ABB RAPID module: Part_8.mod

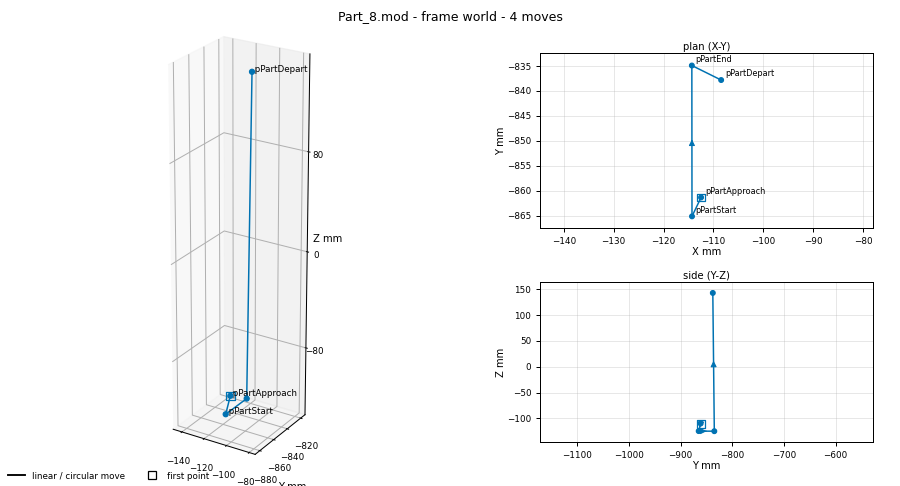
[picture p0: tool path of Part_8.mod in frame world, 4 of 9 moves have a stored position in this frame; points joined in program order, loops and branches not executed]
MODULE Part_8
  ! ------------------------------------------------------------------
  ! Single-part welding template
  !
  ! Purpose:
  !   - Run one part only (no multi-part branching)
  !   - Keep nozzle cleaning and BullsEye tool check available
  !   - Provide a copy/paste starting point for new part files
  !
  ! Dependencies:
  !   - LogicZ (home/safe/pounce positions + rTC2013)
  !   - BE_User1 (BECheckToolb for BullsEye)
  !   - mTSC (optional torch cleaner if you prefer MechCleanGun)
  ! ------------------------------------------------------------------

  PERS bool bUseTorchClean := TRUE;
  PERS bool bUseBullseye := TRUE;

  ! Placeholder weld/seam data for the template. Replace with real values.
  TASK PERS welddata weldPart := [0,0,[1,0,0,0,0,0,0,0,0],[0,0,0,0,0,0,0,0,0]];
  TASK PERS seamdata seamPart := [1,1,[1,0,0,0,0,0,0,0,0],0,0,0,0,0,[0,0,0,0,0,0,0,0,0],0,0,[0,0,0,0,0,0,0,0,0],0,0,[0,0,0,0,0,0,0,0,0],0];

  ! Placeholder targets for the weld path. Replace with taught points.
  CONST robtarget pPartApproach := [[-112.47,-861.36,-110.12],[0.220582,0.688805,-0.67554,-0.143307],[-1,-1,-2,0],[9E+09,9E+09,9E+09,9E+09,9E+09,9E+09]];
  CONST robtarget pPartStart := [[-114.29,-865.15,-124.72],[0.220598,0.688808,-0.675528,-0.143326],[-1,-1,-2,0],[9E+09,9E+09,9E+09,9E+09,9E+09,9E+09]];
  CONST robtarget pPartEnd := [[-114.32,-834.89,-124.92],[0.220557,0.688836,-0.675507,-0.143359],[-1,-1,-2,0],[9E+09,9E+09,9E+09,9E+09,9E+09,9E+09]];
  CONST robtarget pPartDepart := [[-108.44,-837.80,142.79],[0.0521127,0.721407,-0.690258,0.0200149],[-2,-1,-3,0],[9E+09,9E+09,9E+09,9E+09,9E+09,9E+09]];
  PROC RunPart_8()
    TPWrite "Single-part template start";

    ! Optional BullsEye tool check before running a part.
    IF bUseBullseye THEN
      BECheckToolb;
    ENDIF

    ! Optional nozzle cleaning/reaming before the part weld.
    IF bUseTorchClean THEN
      rTC2013;
      ! Alternative: MechCleanGun;  ! From mTSC.mod
    ENDIF

    MoveJ LogicZ::pHomePos, v800, fine, tWeldGun;
    MoveJ LogicZ::pSafeS1, v800, fine, tWeldGun;
    MoveJ LogicZ::pPounceS1, v800, fine, tWeldGun;

    ! ----------------------------------------------------------------
    ! Single-part weld path (edit only the weld start/end points).
    ! ----------------------------------------------------------------
    MoveL pPartApproach, v200, z10, tWeldGun;
    ArcLStart pPartStart, v30, seamPart, weldPart, fine, tWeldGun;
    ArcLEnd pPartEnd, v30, seamPart, weldPart, fine, tWeldGun;
    MoveL pPartDepart, v200, z10, tWeldGun;

    MoveJ LogicZ::pSafeS1, v800, fine, tWeldGun;
    MoveJ LogicZ::pHomePos, v800, fine, tWeldGun;

    TPWrite "Single-part template complete";
  ENDPROC
ENDMODULE
